SUBAPPLICATION Uebung_070_AUI (* WBSD auf UT ausgeben (Adapter Version) *)
  (* Standard: 61499-2; Description: Copyright (c) 2023 Meisterschulen am Ostbahnhof This program and the accompanying materials are made available under the terms of the Eclipse Public License 2.0 which is available at https://www.eclipse.org/legal/epl-2.0/ SPDX-License-Identifier: EPL-2.0 *)
  (* Version 1.0, 2026-04-19, Franz Höpfinger, Meisterschulen am Ostbahnhof, initial API and implementation (Adapter Version of Uebung_070) *)
  PACKAGE Uebungen;
  IMPORT Uebungen::const::UT::TECU::DefaultPool_TECU::NumberVariable_Wheel_based_machine_speed;
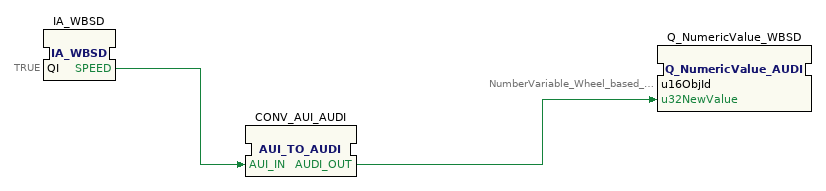
  FBS
    IA_WBSD : isobus::tecu::IA_WBSD(QI := TRUE);
    Q_NumericValue_WBSD : isobus::UT::Q::Q_NumericValue_AUDI(u16ObjId := NumberVariable_Wheel_based_machine_speed);
    CONV_AUI_AUDI : adapter::conversion::unidirectional::AUI_TO_AUDI;
  END_FBS
  ADAPTER_CONNECTIONS
    IA_WBSD.SPEED TO CONV_AUI_AUDI.AUI_IN;
    CONV_AUI_AUDI.AUDI_OUT TO Q_NumericValue_WBSD.u32NewValue;
  END_CONNECTIONS
END_SUBAPPLICATION
